FUNCTION FUN_GetTimestampWithMs : STRING
VAR_INPUT
	stNtTime		:TIMESTRUCT;				// Timestruct with present time
END_VAR
VAR
	sTimestamp		:STRING;					// String to contain timestamp text
	sMiliSec		:STRING;					// Miliseconds in timestamp
END_VAR

// Add data
//sTimeStamp := FUN_GetDate(stNtTime);

// Add time
//sTimestamp := CONCAT(sTimeStamp, ',');
//sTimestamp := CONCAT(sTimeStamp, FUN_GetTime(stNtTime));

// Get mili seconds value 
sMiliSec := '';
sMiliSec := UINT_TO_STRING(stNtTime.wMilliseconds);
IF stNtTime.wMilliseconds < 100 THEN
	sMiliSec := CONCAT(sMiliSec, '0');
	IF stNtTime.wMilliseconds < 10 THEN
		sMiliSec := CONCAT(sMiliSec, '0');
	END_IF
END_IF		

// Create and set timestamp
sTimeStamp := FUN_GetTimestamp(stNtTime);
sTimeStamp := CONCAT(STR1:= sTimeStamp, STR2:= '.'); 
sTimeStamp := CONCAT(STR1:= sTimeStamp, STR2:= sMiliSec); 
	
// Return time stamp
FUN_GetTimestampWithMs := sTimestamp;

END_FUNCTION

(* stored: Version 1.1.0.1, ProductVersion 3.1.4024.12
   POU FUN_GetTimestampWithMs: Id {97361e3e-2f08-4889-9e3e-5e647b319e27}, SpecialFunc None *)
